// TIA Portal V16 export
// export: Created 2023-08-28T09:37:49.6017958Z, ExportSetting WithDefaults, DisplayName Totally Integrated Automation Portal, DisplayVersion V16 Update 6, DisplayName TIA Portal Version Control Interface, DisplayVersion V16 Update 2, DisplayName TIA Portal Openness, DisplayVersion V16 Update 6, DisplayName STEP 7 Professional, DisplayVersion V16 Update 6, DisplayName STEP 7 Safety, DisplayVersion V16, DisplayName WinCC Advanced, DisplayVersion V16 Update 6
DATA_BLOCK "Strategia sterowania POMPOWNIA_DB"   // DB139
AUTHOR : rtecmer
VERSION : 0.1
// stored: AutoNumber true, DBAccessibleFromOPCUA true, InstanceOfName 06_M_Control strategy Pumping station, InstanceOfType FB
"06_M_Control strategy Pumping station"
   // VAR_INPUT
   //    tempStrategia_Pompownia : Int;
   //    "bit_alarm_magistrala _min" : Bool;
   //    bit_off_alarm_magistrala_niskie : Bool;
   // END_VAR
   // VAR_IN_OUT
   //    "Strategia Pompownia" : Int;
   // END_VAR
   // VAR
   //    tmp_on_alarm { ExternalAccessible := 'False'; ExternalVisible := 'False'; ExternalWritable := 'False'} : Bool;
   //    tmp_off_alarm { ExternalAccessible := 'False'; ExternalVisible := 'False'; ExternalWritable := 'False'} : Bool;
   //    memTriger_set_Strategia { ExternalAccessible := 'False'; ExternalVisible := 'False'; ExternalWritable := 'False'} : Bool;
   //    memTriger_reset_Strategia { ExternalAccessible := 'False'; ExternalVisible := 'False'; ExternalWritable := 'False'} : Bool;
   //    test { ExternalAccessible := 'False'; ExternalVisible := 'False'; ExternalWritable := 'False'} : Bool;
   // END_VAR
BEGIN
END_DATA_BLOCK
